Staubli VAL3: loadPage.pgx

program loadPage(string x_sPage, string& x_sItems[])
// load the next page
  local num i
  local string l_sMessage
begin
//  // look if the page libload is correct
//  i=page:libLoad(x_sPage)
//  if i!=0 and i!=11
//    logMsg("INTERFACE:PAGE LIBLOAD "+x_sPage+" result "+toString("",i))
//    popUpMsg("Loading page "+x_sPage+" error CODE "+toString("",i))
//  else
//   // page:sItems=sEvent
//    call page:main()


//  endIf
end
